TYPE ST_Identity_PK2_OUT3 :
STRUCT
	ID	:STRING;
	ReadQuality:STRING;
END_STRUCT
END_TYPE

(* stored: Version 1.1.0.1, ProductVersion 3.1.4024.13
   DUT ST_Identity_PK2_OUT3: Id {bc4ffb99-176d-4aca-9303-b10a8a2674a1} *)
